// SIMATIC S7-200 SMART project (STEP 7-Micro/WIN SMART), CPU CR40

SYMBOL_TABLE 系统符号
Always_On        SM0.0    // 始终接通
END_SYMBOL_TABLE

ORGANIZATION_BLOCK MAIN:OB1
TITLE=程序注释
BEGIN
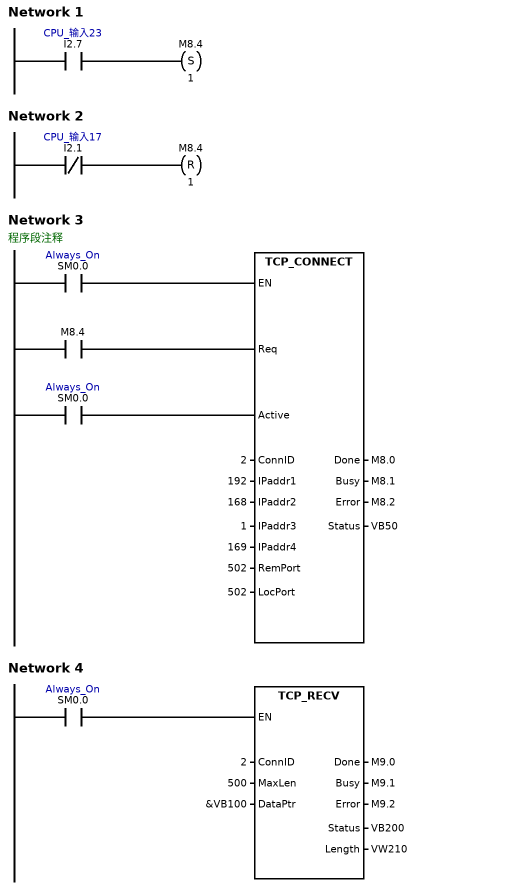
Network 1
LD     CPU_输入23:I2.7
S      M8.4, 1
Network 2
LDN    CPU_输入17:I2.1
R      M8.4, 1
Network 3
// 程序段注释
LD     Always_On:SM0.0
=      L60.0
LD     M8.4
=      L63.7
LD     Always_On:SM0.0
=      L63.6
LD     L60.0
CALL   TCP_CONNECT:SBR1, L63.7, L63.6, 2, 192, 168, 1, 169, 502, 502, M8.0, M8.1, M8.2, VB50
Network 4
LD     Always_On:SM0.0
CALL   TCP_RECV:SBR2, 2, 500, &VB100, M9.0, M9.1, M9.2, VB200, VW210
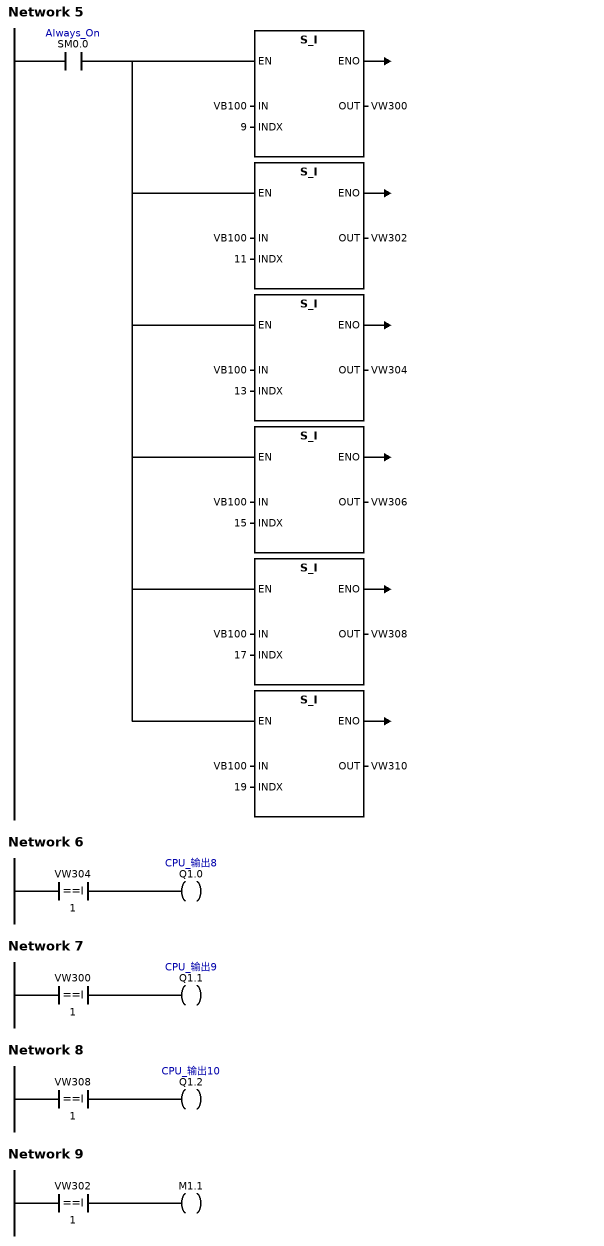
Network 5
LD     Always_On:SM0.0
STI    VB100, 9, VW300
STI    VB100, 11, VW302
STI    VB100, 13, VW304
STI    VB100, 15, VW306
STI    VB100, 17, VW308
STI    VB100, 19, VW310
Network 6
LDW=   VW304, 1
=      CPU_输出8:Q1.0
Network 7
LDW=   VW300, 1
=      CPU_输出9:Q1.1
Network 8
LDW=   VW308, 1
=      CPU_输出10:Q1.2
Network 9
LDW=   VW302, 1
=      M1.1
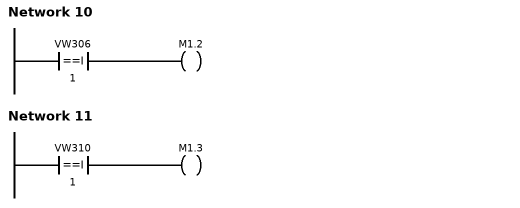
Network 10
LDW=   VW306, 1
=      M1.2
Network 11
LDW=   VW310, 1
=      M1.3
END_ORGANIZATION_BLOCK

// SBR1: protected block, not included

// SBR2: protected block, not included
